% RSLogix 500 project EQU.RSS, saved by version 10.00.00.00 %
PROJECT "UNTITLED"    % processor: Bul.1763 MicroLogix 1100 Series B %

PROGRAM FILES
  LAD 2   2 rungs

DATA FILES
  O0 OUTPUT  4 elements
  I1 INPUT  6 elements
  S2 STATUS  66 elements
  B3 BINARY  1 elements
  T4 TIMER  1 elements
  C5 COUNTER  1 elements
  R6 CONTROL  1 elements
  N7 INTEGER  1 elements
  F8 FLOAT  1 elements

LADDER 2
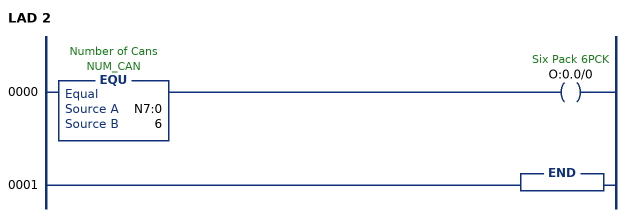
% Rung: 0 %
SOR EQU N7:0 6 OTE O:0.0/0 EOR
%   N7:0  NUM_CAN  "Number of Cans" %
%   O:0.0/0  6PCK  "Six Pack" %
% Rung: 1 %
SOR END EOR

OTHER DOCUMENTED ADDRESSES
  C5:0  MTR_STR  "Motor Starts"
  I:0.0/1  MTR_STAT  "Motor Status"
  T4:0  MTR_TMR  "Motor Timer"

DATA TABLE (non-zero values as saved)
DATA T4
% .PRE .ACC %
% T4:0 % 8 0
DATA C5
% .PRE .ACC %
% C5:0 % 1000 -32768
DATA N7
% N7:0 % 3
